(* CoDeSys 2.3.9.50 project: counter.pro *)
(* Libraries: STANDARD.LIB 5.6.98 11:03:02 *)

(* Task configuration *)
TASK Standard (PRIORITY := 0, INTERVAL := T#10ms);
	MAIN
END_TASK

(* Global variable list: Global_Variables *)
VAR_GLOBAL
	Knop1 : BOOL;
	Knop2: BOOL;
	Lamp1 : BOOL;


END_VAR

(* Global variable list: TwinCAT_Configuration *)
(* Generated automatically by TwinCAT - (read only) *)
VAR_CONFIG
	test.bTestInput AT %IX0.0 : BOOL;	(*  ~ {LinkedWith:TIID^Device 1 (EtherCAT)^Term 19 (EK1100)^Term 20 (EM7004)^DI Inputs^Input^test.bTestInput} *)
	test.bTestInput2 AT %IX4.0 : BOOL;
	test.bTestOutput AT %QX0.0 : BOOL;
END_VAR

(* POU MAIN, ST *)
PROGRAM MAIN
VAR

END_VAR
count() ;
END_PROGRAM

(* POU count, ST *)
PROGRAM count
VAR
	count: INT;

	counter: CTU;
END_VAR
counter(
	CU:=Knop1 ,
	RESET:= , 
	PV:= , 
	Q=> ,
	CV=>count );
END_PROGRAM

(* POU Blinker, ST *)
PROGRAM Blinker
VAR

	tTijdAan : TIME;
	tTijdUit : TIME;
	Lamp1: BOOL;
	Knop1 : BOOL;
	Knop2 : BOOL;
	Vrijgave : BOOL;
	Blink : BOOL;



	Lamp1_aan: BOOL;
	Lamp1_uit: BOOL;


	Lamp1Uit: BOOL;

	rtFallingEdge : F_TRIG;
	pulse1 : TP;
	pulse2 : TP;


END_VAR
tTijdAan := T#1S;
tTijdUit :=T#1S;


Lamp1_aan := Knop1 AND NOT Vrijgave;


pulse1(IN:=Lamp1_aan , PT:=tTijdAan , Q=>Lamp1);

rtFallingEdge(CLK:=Lamp1 , Q=>Lamp1_uit );


pulse2(IN:=Lamp1_uit , PT:=tTijdUit , Q=>Vrijgave);
END_PROGRAM

(* POU test, ST *)
PROGRAM test

VAR

	bTest: BOOL;
	bTestInput          AT %I*:        BOOL;
	bTestInput2          AT %I*:        BOOL;
	bTestOutput       AT %Q*:        BOOL;

	Knop1 : BOOL;
	Knop2 : BOOL;
	Knop3 : BOOL;
	Knop4 : BOOL;

	Lamp1 : BOOL;
	Lamp2 : BOOL;
	Lamp3 : BOOL;
	Lamp4 : BOOL;

	Knop1_old : BOOL;

	tT1 : TOF;


END_VAR
bTest := TRUE ;




tT1(IN:=Knop1 , PT:=T#1s , Q=>Lamp1 );
END_PROGRAM
